Universal Robots PolyScope program: Levanic_reconstruction_communication.urp

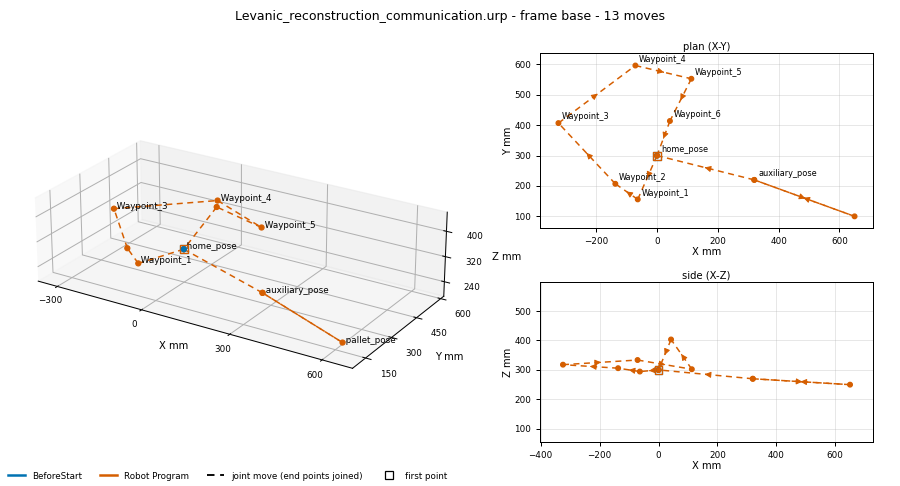
[picture p0: tool path of Levanic_reconstruction_communication.urp in frame base, 13 of 16 moves have a stored position in this frame; points joined in program order, loops and branches not executed]
Program Levanic_reconstruction_communication (installation=Levanic directory=/programs/Levanic createdIn=5.9.5.1031259 lastSavedIn=5.9.5.1031259 robotSerialNumber=20215500386)
Calibrated DH parameters: a=[0.000206, -0.276434, -0.392186, 0.000086, 0.00001, 0]; d=[0.162469, -361.266131, 361.052801, 0.346944, 0.099711, 0.099657]; alpha=[1.571293, -0.000893, 0.005969, 1.570168, -1.570592, 0]; deltaTheta=[0, 0.862555, -0.865797, 0.003247, 0, 0]
BeforeStart
  Popup Message (haltProgram=false message=Start program? inputType=Text)
  MoveJ speed 60 deg/s, acceleration 80 deg/s^2 (useActiveTCP=true) feature=Base
    Waypoint home_pose: TCP in base x=0 y=300 z=300 mm, rx=0 ry=0 rz=0 rad; joints [-116.503, -116.854, 93.746, -66.881, 270.323, -26.555] deg; TCP offset x=0 y=0 z=295 mm, rx=3.1416 ry=0 rz=0 rad
  sending_str := ""
  received_float := 0
  Script: socket_state=socket_open("192.168.40.191", 34500)
Robot Program (runOnlyOnce=false)
  Wait Sleep waitTime=0.1
  Call ReceiveStringData
  If received_str≟"RECONSTRUCT"
    Wait Sleep waitTime=2
    MoveJ speed 60 deg/s, acceleration 80 deg/s^2 (useActiveTCP=true) feature=Base
      Waypoint home_pose: TCP in base x=0 y=300 z=300 mm, rx=0 ry=0 rz=0 rad; joints [-116.503, -116.854, 93.746, -66.881, 270.323, -26.555] deg
      Waypoint Waypoint_1: TCP in base x=-63.44 y=155.846 z=294.496 mm, rx=-0.0485 ry=-0.1895 rz=1.1644 rad; joints [-90.837, -134.73, 101.917, -60.837, 260.377, -68.146] deg; TCP offset x=0 y=0 z=295 mm, rx=3.1416 ry=0 rz=0 rad
      Call SendRobotAndReceivePCData
      Waypoint Waypoint_2: TCP in base x=-137.151 y=207.093 z=305.88 mm, rx=-0.3526 ry=-0.3014 rz=1.2112 rad; joints [-59.86, -104.111, 86.183, -54.088, 252.726, -37.758] deg
      Call SendRobotAndReceivePCData
      Waypoint Waypoint_3: TCP in base x=-324.365 y=406.851 z=317.818 mm, rx=-0.0387 ry=-0.2544 rz=-0.1349 rad; joints [-58.241, -72.714, 50.223, -57.116, 259.781, 40.36] deg
      Call SendRobotAndReceivePCData
      Waypoint Waypoint_4: TCP in base x=-71.151 y=596.288 z=333.601 mm, rx=0.2008 ry=-0.1805 rz=-1.6708 rad; joints [-87.022, -70.039, 46.416, -65.64, 256.59, 99.22] deg
      Call SendRobotAndReceivePCData
      Waypoint Waypoint_5: TCP in base x=112.997 y=552.743 z=302.376 mm, rx=-0.1305 ry=0.2618 rz=-1.9426 rad; joints [-125.637, -83.568, 68.229, -73.088, 284.46, 76.094] deg
      Call SendRobotAndReceivePCData
      Waypoint Waypoint_6: TCP in base x=42.484 y=413.785 z=403.334 mm, rx=0.3404 ry=0.5736 rz=-1.7846 rad; joints [-148.142, -128.39, 95.638, -72.848, 299.953, 51.576] deg
      Call SendRobotAndReceivePCData
      Waypoint home_pose: TCP in base x=0 y=300 z=300 mm, rx=0 ry=0 rz=0 rad; joints [-116.503, -116.854, 93.746, -66.881, 270.323, -26.555] deg; TCP offset x=0 y=0 z=295 mm, rx=3.1416 ry=0 rz=0 rad
    Call SendFinishedData
  ElseIf received_str≟"HANDLE"
    Call SendRobotData
    Call ReceivePoseData
    appr_trans_vec := translation_vec
    appr_rot_vec := rotation_vec
    Call SendRobotData
    Call ReceivePoseData
    grab_trans_vec := translation_vec
    grab_rot_vec := rotation_vec
    Call SendRobotData
    Call ReceiveFloatData
    gripper_width := received_float
    calc_grip_width := (gripper_width*1000+23)/3.3
    If appr_trans_vec[2]≥-0.02 and grab_trans_vec[2]≥-0.02
      approach_pose := p[appr_trans_vec[0],appr_trans_vec[1],appr_trans_vec[2],appr_rot_vec[0],appr_rot_vec[1],appr_rot_vec[2]]
      grabbing_pose := p[grab_trans_vec[0],grab_trans_vec[1],grab_trans_vec[2],grab_rot_vec[0],grab_rot_vec[1],grab_rot_vec[2]]
      Script: rq_move_and_wait_mm(calc_grip_width)
      MoveL speed 150 mm/s, acceleration 600 mm/s^2 (useActiveTCP=true) feature=Base
        Waypoint Waypoint (Variable): variable=approach_pose
      MoveL speed 50 mm/s, acceleration 200 mm/s^2 (useActiveTCP=true) feature=Base
        Waypoint Waypoint (Variable): variable=grabbing_pose
      URCap Gripper (Robotiq_Grippers, Robotiq Inc.) dataModel(position=100.0, force=20.0, speed=50.0, positionInDouble=100.0, forceInDouble=20.0, speedInDouble=50.0, slaveIds=[9], blocking=true)
      MoveL speed 150 mm/s, acceleration 600 mm/s^2 (useActiveTCP=true) feature=Base
        Waypoint Waypoint (Variable): variable=approach_pose
      MoveJ speed 60 deg/s, acceleration 80 deg/s^2 (useActiveTCP=true) feature=Base
        Waypoint auxiliary_pose: TCP in base x=320 y=220 z=270 mm, rx=0 ry=0 rz=0 rad; joints [-165.667, -105.814, 91.916, -76.091, 270.332, -75.671] deg; TCP offset x=0 y=0 z=295 mm, rx=3.1416 ry=0 rz=0 rad
        Waypoint pallet_pose: TCP in base x=650 y=100 z=250 mm, rx=0.1275 ry=-0.6489 rz=-1.008 rad; joints [-174.65, -93.281, 103.99, -134.397, 256.219, -28.771] deg; TCP offset x=0 y=0 z=295 mm, rx=3.1416 ry=0 rz=0 rad
      Script: rq_move_and_wait_mm(calc_grip_width)
      URCap Gripper (Robotiq_Grippers, Robotiq Inc.) dataModel(position=100.0, force=20.0, speed=50.0, positionInDouble=100.0, forceInDouble=20.0, speedInDouble=50.0, slaveIds=[9], blocking=true)
      MoveJ speed 60 deg/s, acceleration 80 deg/s^2 (useActiveTCP=true) feature=Base
        Waypoint auxiliary_pose: TCP in base x=320 y=220 z=270 mm, rx=0 ry=0 rz=0 rad; joints [-165.667, -105.814, 91.916, -76.091, 270.332, -75.671] deg; TCP offset x=0 y=0 z=295 mm, rx=3.1416 ry=0 rz=0 rad
        Waypoint home_pose: TCP in base x=0 y=300 z=300 mm, rx=0 ry=0 rz=0 rad; joints [-116.503, -116.854, 93.746, -66.881, 270.323, -26.555] deg; TCP offset x=0 y=0 z=295 mm, rx=3.1416 ry=0 rz=0 rad
      Call SendFinishedData
    Else 
      Popup Message (haltProgram=false message=Approaching or grabbing height is lower than ground-level! inputType=Text)
SubProgram -> SendFinishedData
SubProgram -> SendRobotData
SubProgram -> SendRobotAndReceivePCData
SubProgram -> ReceiveStringData
SubProgram -> ReceiveFloatData
SubProgram -> ReceivePoseData
SubProgram ReceiveStringData (keepSynchronizedWithDisk=false)
  received_str := socket_read_string()
SubProgram SendRobotAndReceivePCData (keepSynchronizedWithDisk=false)
  Script: socket_send_string("ROBOT READY")
  received_pc := socket_read_string()
  Loop While (checkContinuously=false) expression=received_pc≠"PC READY"
    received_pc := socket_read_string()
SubProgram SendFinishedData (keepSynchronizedWithDisk=false)
  Script: socket_send_string("FINISHED")
SubProgram SendRobotData (keepSynchronizedWithDisk=false)
  Script: socket_send_string("ROBOT READY")
SubProgram ReceivePoseData (keepSynchronizedWithDisk=false)
  rec_raw_pose := socket_read_ascii_float(6)
  If rec_raw_pose[0]≟6
    translation_vec := [rec_raw_pose[1], rec_raw_pose[2], rec_raw_pose[3]]
    rotation_vec := [rec_raw_pose[4], rec_raw_pose[5], rec_raw_pose[6]]
SubProgram ReceiveFloatData (keepSynchronizedWithDisk=false)
  rec_raw_float := socket_read_ascii_float(1)
  If rec_raw_float[0]≟1
    received_float := rec_raw_float[1]
